// TIA Portal V17 export
// export: Created 2025-03-07T09:17:30.5446536Z, ExportSetting WithDefaults, DisplayName Totally Integrated Automation Portal, DisplayVersion V17 Update 8, DisplayName TIA Portal Openness, DisplayVersion V17 Update 8, DisplayName TIA Portal Version Control Interface, DisplayVersion V17, DisplayName SINAMICS Startdrive Advanced, DisplayVersion V17 SP2, DisplayName SINAMICS Startdrive G110M, G120, G120C, G120D, G120P, G115D, DisplayVersion V17 SP2, DisplayName SINAMICS Startdrive G130, G150, S120, S150, SINAMICS MV, S210, DisplayVersion V17 SP2, DisplayName STEP 7 Professional, DisplayVersion V17 Update 8, DisplayName SINUMERIK ONE STEP 7 Toolbox, DisplayVersion V17 Update 12, DisplayName SINUMERIK 840D sl STEP 7 Toolbox, DisplayVersion V17 Update 12, DisplayName STEP 7 Safety, DisplayVersion V17 Update 6, DisplayName WinCC Advanced, DisplayVersion V17 Update 8
DATA_BLOCK "DB318_CH8_PROGRAM_SELECTION"   // DB318
{ DB_Accessible_From_OPC_UA := 'FALSE' }
AUTHOR : ETXETAR
VERSION : 1.0
// stored: AutoNumber false, DBAccessibleFromOPCUA false, DBAccessibleFromWebserver true, InstanceOfName FB311_CHANNEL_PROGRAM_SELECTION, InstanceOfType FB
"FB311_CHANNEL_PROGRAM_SELECTION"
   // VAR_INPUT
   //    REQUEST : Bool;
   // END_VAR
   // VAR_OUTPUT
   //    ALARM : Bool;
   // END_VAR
   // VAR_IN_OUT
   //    channelDB : "LBP_typeChanX";
   // END_VAR
   // VAR RETAIN
   //    interlocksDB { S7_SetPoint := 'True'} : "CNC_PLC_INT_CH";
   //    FB7_INSTANCE { S7_SetPoint := 'True'} : "LBP_ReqPIService";
   // END_VAR
BEGIN
   interlocksDB.PName := '_N_CH8_MEASURE_MPF';
   interlocksDB.Path := '/_N_WKS_DIR/_N_CH_8_WPD';
END_DATA_BLOCK
